TYPE ST_ItemTemporary :
STRUCT
	Item	: ST_Item;
	Counts	: UDINT;
END_STRUCT
END_TYPE

(* stored: Version 1.1.0.1, ProductVersion 3.1.4024.4
   DUT ST_ItemTemporary: Id {49f554c6-7765-4710-a482-c50efa83427f} *)
